(*	
*)
FUNCTION_BLOCK FB_MotionlinxAI_Axis EXTENDS FB_ComponentBase //IMPLEMENTS I_MotionlinxAI_Axis
VAR
	//Controller Status	

	_Controller_Sts	:ST_Controller_Status;
	
	
	
//Inputs
	iServoState	AT%I* : SINT;	
	iPosition 		AT%I* : INT;
	iDiagnostics	AT%I* : INT;
	
	//Speed Limits//
	uMaxSpeed (*AT%I**) : UINT;		//ACTION - IS this from the drive??????
	uMinSpeed : UINT;

//Output
	oMotorControl	AT%Q* : SINT;
	oMotorSpeed		AT%Q* : INT;
	oMotorBrakeMode	AT%Q* : SINT := 2;
	oMotorAccel		AT%Q* : INT;
	oMotorDecel	AT%Q* : INT;
	oServoPos		AT%Q* : INT;
	//Servo Setting//	
	bSetServo : BOOL;
	bHomed : BOOL;
	


	// Internal variables
	//Run Motor//	
	bEnabled : BOOL;
	bRunMotor : BOOL;
	nRequestedSpeed : UINT;


//	iSensors	:INT;
	//Error Resetting//
	//bError : BOOL;
	tpErrorReset : TP;
	//Motor Status//
	eMotorStatus: MotionlinxAI_Motor_Status;
	eErrorRecord : MotionlinxAI_Error_States;
	eMotionlinxAIState : MotionlinxAI_States;
	Main_Sensor	: BOOL;
	Aux_Sensor	: BOOL;
	
	eError : MotionlinxAI_Error_States;
	
	bMotorExpected : BOOL;
	bMotorDisconnected: BOOL;
	
	iPreviousPosition	:int;

	// Timer for Extend/Retract
	tonAxisStopped	:ton:=(PT:=T#0.5S);
	bAxis_Stopped	:BOOL;

	//HMI 
	MotionlinxAI_HMI : ST_MotionlinxAI_Axis_HMI;
	
	iCounter	:int;
END_VAR

PROPERTY Acceleration : int
SET
oMotorAccel	:= Acceleration;
//Recipe.Axis.Acceleration := Acceleration;
END_SET
END_PROPERTY

ACTION Astop:
//oMotorLControl.0 := FALSE;
//oMotorRControl.0 := FALSE;
END_ACTION

PROPERTY Controller_Sts : ST_Controller_Status
SET
_Controller_Sts	:=Controller_Sts;
END_SET
END_PROPERTY

METHOD PROTECTED CreateEvents
VAR_INPUT
END_VAR
SUPER^.CreateEvents();
END_METHOD

METHOD CyclicLogic
iCounter	:= iCounter +1;
errorCheck();


Main_Sensor	:= _Controller_Sts.Sensors.4;		//ACTION Need logic to swap sensors dependinf on input group 1 or 2 Main aux
Aux_Sensor	:= _Controller_Sts.Sensors.0;

//
//ACTION Need logic to swap sensors dependinf on input group 1 or 2 Main aux

//////////Set State//////////
//////////Set State//////////
IF _Error THEN
	eMotionlinxAIState := MotionlinxAI_States.ERROR;
ELSIF bSetServo  THEN
	IF bHomed THEN
		IF eMotorStatus > MotionlinxAI_Motor_Status.MOTOR_NOT_RUNNING_UNBRAKED THEN
			eMotionlinxAIState := MotionlinxAI_States.RUNNING;
		ELSIF eMotorStatus <= MotionlinxAI_Motor_Status.MOTOR_NOT_RUNNING_UNBRAKED  THEN
			eMotionlinxAIState := MotionlinxAI_States.STOPPED;
		END_IF
	ELSE
		eMotionlinxAIState := MotionlinxAI_States.HOMING;
	END_IF
ELSE
	IF eMotorStatus > MotionlinxAI_Motor_Status.MOTOR_NOT_RUNNING_UNBRAKED  THEN
		eMotionlinxAIState := MotionlinxAI_States.RUNNING;
	ELSIF eMotorStatus <= MotionlinxAI_Motor_Status.MOTOR_NOT_RUNNING_UNBRAKED  THEN
		eMotionlinxAIState := MotionlinxAI_States.STOPPED;
	END_IF
END_IF



uMinSpeed := 15+uMaxSpeed/100;


//////////Motor Status//////////
IF iDiagnostics.0 AND iDiagnostics.1 THEN
	eMotorStatus := MotionlinxAI_Motor_Status.MOTOR_NOT_RUNNING_UNBRAKED;
ELSIF iDiagnostics.0 AND NOT iDiagnostics.1 THEN
	eMotorStatus := MotionlinxAI_Motor_Status.MOTOR_RUNNING_CCW;
ELSIF NOT iDiagnostics.0 AND iDiagnostics.1 THEN
	eMotorStatus := MotionlinxAI_Motor_Status.MOTOR_RUNNING_CW;
ELSIF NOT iDiagnostics.0 AND NOT iDiagnostics.1 THEN
	eMotorStatus := MotionlinxAI_Motor_Status.MOTOR_NOT_RUNNING_BRAKED;
END_IF;

//////////Stop On Disable//////////
IF NOT bEnabled THEN
	oMotorDecel := 500;	
	oMotorControl.0 := FALSE;
//ELSE
//	oMotorDecel := 500;
END_IF;

//////////Set Speeds//////////
oMotorSpeed := LIMIT(UINT_TO_INT(uMinSpeed),UINT_TO_INT(nRequestedSpeed),UINT_TO_INT(uMaxSpeed));

tonAxisStopped(IN:= iPosition=iPreviousPosition, Q => bAxis_Stopped);
iPreviousPosition	:= iPosition;

//One shot the requests
//Extend_RTRIG(CLK := _ExtendRequest);
//Retract_RTRIG(CLK := _RetractRequest);

////Handle Extend
//IF Extend_RTRIG.Q THEN
////	Output			:= TRUE;
//	_Extending		:= TRUE;
//	_Retracting		:= FALSE;
//	_Retracted		:= FALSE;
//	_RetractRequest := FALSE;
//END_IF

////Handle Retract
//IF Retract_RTRIG.Q THEN
////	Output		   := FALSE;
//	_Extending	   := FALSE;
//	_Retracting	   := TRUE;
//	_Extended	   := FALSE;
//	_ExtendRequest := FALSE;
//END_IF

////Handle the time to Extend/Retract
//Extend_TON(IN := _Extending, PT := LREAL_TO_TIME(_ExtendTime));
//Retract_TON(IN := _Retracting, PT := LREAL_TO_TIME(_RetractTime));
//IF Extend_TON.Q THEN
//	_Extended  := TRUE;
//	_Extending := FALSE;
//END_IF

//IF Retract_TON.Q THEN
//	_Retracted	:= TRUE;
//	_Retracting := FALSE;
//END_IF

SUPER^.CyclicLogic();
END_METHOD

PROPERTY Deceleration : int
SET
oMotorDecel	:= Deceleration;
END_SET
END_PROPERTY

METHOD Disable : BOOL
(*BRAKING MODES:
	0 : NORMAL - HOLDS IN PLACE BY SHORTING WINDINGS
	1 : FREE - NOT HELD IN PLACE
	2 : SERVO - MAINTAINS POSITION BASED ON HALLS EFFECT SENSOR*)
//oMotorDecel := 500;
bEnabled := FALSE;
END_METHOD

METHOD EmergencyStop : BOOL
(*BRAKING MODES:
	0 : NORMAL - HOLDS IN PLACE BY SHORTING WINDINGS
	1 : FREE - NOT HELD IN PLACE
	2 : SERVO - MAINTAINS POSITION BASED ON HALLS EFFECT SENSOR*)
oMotorDecel:= 1;
oMotorControl.0 := FALSE;
bEnabled := FALSE;
oMotorBrakeMode := 0;
END_METHOD

METHOD Enable : BOOL
VAR_INPUT
//	Acceleration	:INT;	//Should not be here, but part of recipe
END_VAR
(*BRAKING MODES:
	0 : NORMAL - HOLDS IN PLACE BY SHORTING WINDINGS
	1 : FREE - NOT HELD IN PLACE
	2 : SERVO - MAINTAINS POSITION BASED ON HALLS EFFECT SENSOR*)
bEnabled := TRUE;
//oMotorAccel	:= Acceleration;
//oMotorControl.0 := TRUE;
//oMotorBrakeMode  := 2;
END_METHOD

PROPERTY Enabled : BOOL
GET
Enabled := bEnabled;
END_GET
END_PROPERTY

ACTION errorCheck:
//oClearMotorError := 0;	//Action. this goes to the contrroller and that sends the reset requests
IF  iDiagnostics.5  THEN
	eError := MotionlinxAI_Error_States.MOTOR_BOARD_OVERHEAT;
(*ELSIF iDiagnosticsL.6  THEN
	eErrorLeft := MotionlinxAI_Error_States.MOTOR_OVERVOLTAGE;
ELSIF iDiagnosticsL.7  THEN
	eErrorLeft := MotionlinxAI_Error_States.MOTOR_UNDERVOLTAGE;*)
ELSIF iDiagnostics.8  THEN
	eError := MotionlinxAI_Error_States.MOTOR_OVERHEATED;
(*ELSIF iDiagnosticsL.9  THEN
	eErrorLeft := MotionlinxAI_Error_States.MOTOR_MAX_TORQUE;*)
ELSIF iDiagnostics.10  THEN
	eError := MotionlinxAI_Error_States.MOTOR_SHORT_CIRCUIT;
ELSIF iDiagnostics.11  THEN
	eError := MotionlinxAI_Error_States.MOTOR_NOT_CONNECTED;
ELSIF iDiagnostics.12  THEN
	eError := MotionlinxAI_Error_States.MOTOR_OVERLOADED;
ELSIF iDiagnostics.13  THEN
	eError := MotionlinxAI_Error_States.MOTOR_STALLED;
ELSIF iDiagnostics.14  THEN
	eError := MotionlinxAI_Error_States.MOTOR_HALL_SENSOR;
ELSE
	eError := MotionlinxAI_Error_States.NO_ERROR;
END_IF;



bMotorDisconnected := eError = MotionlinxAI_Error_States.MOTOR_NOT_CONNECTED;

IF eError <> MotionlinxAI_Error_States.NO_ERROR  OR eError = MotionlinxAI_Error_States.MOTOR_UNDERVOLTAGE  THEN
	IF (bMotorDisconnected AND NOT bMotorExpected)  THEN
		_Error := FALSE;
	ELSE
		_Error := TRUE;
		eError := eError;
	
			
//		IF oClearMotorError = 0 THEN
//			oClearMotorError := 1;
//		ELSIF oClearMotorError = 1 THEN
//			oClearMotorError := 0;
//		END_IF;
	END_IF

ELSE
	_Error := FALSE;
END_IF;
END_ACTION

PROPERTY HasFault : BOOL
GET
HasFault := eMotionlinxAIState < MotionlinxAI_States.HOMING;// or bCommunicationsFailed;
END_GET
END_PROPERTY

METHOD PROTECTED HMICommunication
VAR_INPUT
END_VAR
SUPER^.HMICommunication();

//Handle the requests to extend and retract
IF ComponentBase_HMI.Status.HMIControlAvailable THEN
	IF MotionlinxAI_HMI.Command.Extend THEN
//		Extend();
	ELSIF MotionlinxAI_HMI.Command.Retract THEN
//		Retract();
	END_IF
END_IF

//Update HMI status info
//Cylinder_HMI.Status.Extended	:= _Extended;
//Cylinder_HMI.Status.Extending	:= _Extending;
//Cylinder_HMI.Status.Retracted	:= _Retracted;
//Cylinder_HMI.Status.Retracting	:= _Retracting;
//Cylinder_HMI.Config.ExtendTime	:= _ExtendTime;
//Cylinder_HMI.Config.RetractTime := _RetractTime;
END_METHOD

//! @summary Basic component initialization logic
METHOD PROTECTED Initialize : BOOL;

//! @description This method is called by <c>CyclicLogic()</c> as required



//Set the cylinder to retracted
//oMotorAccel	:= 500;		//From recipe value here
//IF Output THEN
//	_Extended  := TRUE;
//	_Retracted := FALSE;
//ELSE
//	_Extended  := FALSE;
//	_Retracted := TRUE;
//END_IF



//Call base class Initialize
Initialize := SUPER^.Initialize();
END_METHOD

PROPERTY IsReady : BOOL
GET
IsReady := eMotionlinxAIState > MotionlinxAI_States.HOMING;
END_GET
END_PROPERTY

PROPERTY MaxSpeed : uint
SET
uMaxSpeed	:= MaxSpeed;
END_SET
END_PROPERTY

METHOD PROTECTED Monitoring
VAR_INPUT
END_VAR
_Busy	 := NOT Stopped;//MotionlinxAI_Motor_Status:=3 OR MotionlinxAI_Motor_Status:=4 ;
_Error	 := eError>0 OR eMotionlinxAIState < MotionlinxAI_States.HOMING;;
_ErrorID := eError;
SUPER^.Monitoring();
END_METHOD

PROPERTY MotorDisconnected : bool
GET
MotorDisconnected	:= bMotorDisconnected;
END_GET
END_PROPERTY

METHOD Start : BOOL
VAR_INPUT
END_VAR
IF bEnabled THEN 
	oMotorControl.0 := TRUE;
	oMotorBrakeMode  := 2;
END_IF
END_METHOD

METHOD Stop
VAR_INPUT
END_VAR
oMotorControl.0 := FALSE;
oMotorBrakeMode := 2;
END_METHOD

PROPERTY Stopped : bool
GET
Stopped	:= bAxis_Stopped;
END_GET
END_PROPERTY

PROPERTY Velocity : int
SET
nRequestedSpeed	:= Velocity;
//Recipe.Axis.Acceleration := Acceleration;
END_SET
END_PROPERTY

END_FUNCTION_BLOCK

(* stored: Version 1.1.0.1, ProductVersion 3.1.4024.16
   POU FB_MotionlinxAI_Axis: Id {84bed10e-2014-44a4-86fd-506ddbbef3d2}, SpecialFunc None
   Folder I_ComponentBase: Id {564bca5b-815b-4420-a3bf-27ca975dea8a}
   Folder I_CyclicFB: Id {e674dbf9-cf5e-458c-94b6-d3dcdd89cb73}
   Folder I_MotionlinxAI_Axis: Id {03e0a6a9-6324-40f7-9830-f10137e10bd5}
   Property Acceleration: Id {d91cb6df-d18c-43c9-aff0-8443b35bbdf5}
   Set Set: Id {65466805-8aa0-49a3-8df9-6cdf97f534be}
   Action Astop: Id {d5c43eb1-1d38-4e44-8bc2-00e2b5bb6fa6}
   Property Controller_Sts: Id {88f38349-94a3-422a-9722-22b42b0cdd49}
   Set Set: Id {4b928b3d-76ba-4673-b0cf-fba390a3ca23}
   Method CreateEvents: Id {e0f8766d-dc7c-457b-9343-3c71d71e0eda}
   Method CyclicLogic: Id {39eda1b4-62f4-459e-961e-ef10a5bb498b}
   Property Deceleration: Id {1a153ede-59af-4d81-b343-2a04bc992805}
   Set Set: Id {bdadbec4-d50b-4d0a-879d-5fa57e176119}
   Method Disable: Id {1d453f6e-3687-4412-ae4d-5e48024c3ad0}
   Method EmergencyStop: Id {8591e24a-3de3-441d-a69f-a1e1e7e28cb2}
   Method Enable: Id {e5af88bd-408e-4e07-8d90-41c559ff9446}
   Property Enabled: Id {584b0cad-97bc-486f-baa5-ad501022e39e}
   Get Get: Id {dc9be4db-7694-42dc-a45a-bd0ea8a3eb63}
   Action errorCheck: Id {5b89c9f1-6a13-405d-9c8a-b081e6c5d852}
   Property HasFault: Id {97dbf5df-348c-4c25-b4a9-4d7e37e13d72}
   Get Get: Id {95336fac-c4c0-44b6-ba08-00eb0e158768}
   Method HMICommunication: Id {249af752-b6a6-44b3-8c53-18dccc43eb48}
   Method Initialize: Id {07e4833f-62d9-4f46-89f6-ec9a6c2d1480}
   Property IsReady: Id {b384d1c3-b2d2-456b-9703-0b46c4cb2e78}
   Get Get: Id {e3ebbcf6-ec46-4dbe-bfbe-160047b83ec7}
   Property MaxSpeed: Id {3e716af1-c7b7-440a-84a8-8ae7c2314148}
   Set Set: Id {5819c363-d272-4380-9be4-da5affa2a8eb}
   Method Monitoring: Id {35f17985-3d10-4a38-b8a2-8d66a31a369c}
   Property MotorDisconnected: Id {056db5c2-f9f1-4268-a28d-dc0353d09bbb}
   Get Get: Id {0231605c-467e-421a-b54a-25eb681f92ab}
   Method Start: Id {66c34b9d-4bd7-4fcb-8bfe-152fa560519d}
   Method Stop: Id {1ebcc6dd-875d-4fcf-a089-89f14e84fd33}
   Property Stopped: Id {e3cdb5b7-236b-4b6e-b047-4981e2a4591f}
   Get Get: Id {d9788d61-7d76-4502-86e3-333f66cfe51c}
   Property Velocity: Id {cbbaa72b-1a2b-4384-8fee-2c5410c0803a}
   Set Set: Id {aa82b17e-d9c0-4f75-83d6-d86f4db44c95} *)
